Yaskawa INFORM job: R2-MOVE.JBI

/JOB
//NAME R2-MOVE
//POS
///NPOS 6,0,0,0,0,0
///TOOL 1
///POSTYPE PULSE
///PULSE
C00000=-6022,-65326,-52845,3,-2902,-16
C00001=-62782,-65326,-52845,3,-2902,-16
C00002=-62782,-65326,-98385,3,-2902,-16
C00003=38066,-65326,-98385,3,-2902,-16
C00004=38066,-65326,-48193,3,-2902,-16
C00005=-25294,-65326,-48193,3,-2902,-16
//INST
///DATE 2023/02/06 16:50
///ATTR SC,RW
///GROUP1 RB2
NOP
MOVJ C00000 VJ=10.00
MOVL C00001 V=83.3
MOVL C00002 V=83.3
MOVL C00003 V=83.3
MOVL C00004 V=83.3
MOVL C00005 V=83.3
END
